FUNCTION_BLOCK SUB_UINT (* IEC 61131-3 UINT Subtraction *)
  (* Standard: 61131-3 *)
  (* Version 0.0, 2006-09-11, JHC, Holobloc Inc *)
  (* Compiler header: package fb.rt.plc.math; *)
  (* Compiler classdef: (Math.max(0, IN1 - IN2 )) *)
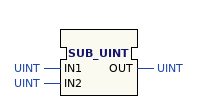
  VAR_INPUT
    IN1 : UINT; (* Minuend *)
    IN2 : UINT; (* Subtrahend *)
  END_VAR
  VAR_OUTPUT
    OUT : UINT; (* Difference *)
  END_VAR
END_FUNCTION_BLOCK
